{attribute 'linkalways'} 
{attribute 'no_explicit_call' := 'This FB is a CLASS and must be accessed using methods or properties'}
{attribute 'enable_dynamic_creation'}
FUNCTION_BLOCK RetrieveNodeContentValue IMPLEMENTS I_GraphVisitor, I_NodeVisitor, I_ContentVisitor
VAR
	graphUuid : T_MAXSTRING;
	nodeId : T_MAXSTRING;
	contentName : T_MAXSTRING;
	serializer : I_Serializer;
	_done : BOOL;
	_error : BOOL;
	_errorMessage : T_MAXSTRING;
END_VAR

PROPERTY PUBLIC Done : BOOL
GET
Done := _done;
END_GET
END_PROPERTY

PROPERTY PUBLIC Error : BOOL
GET
Error := _error;
END_GET
END_PROPERTY

PROPERTY PUBLIC ErrorMessage : T_MAXSTRING
GET
ErrorMessage := _errorMessage;
END_GET
END_PROPERTY

METHOD PUBLIC Initialize
VAR_INPUT
	GraphUuid : T_MAXSTRING;
	NodeId : T_MAXSTRING;
	ContentName : T_MAXSTRING;
	Serializer : I_Serializer;
END_VAR
THIS^.graphUuid := GraphUuid;
THIS^.nodeId := NodeId;
THIS^.contentName := ContentName;
THIS^.serializer := Serializer;
END_METHOD

METHOD PRIVATE LogInvalidContentNameError
VAR_INPUT
END_VAR
_errorMessage := 'Invalid Content Name';
_error := TRUE;
END_METHOD

METHOD PRIVATE LogInvalidNodeIdError
VAR_INPUT
END_VAR
_errorMessage := 'Invalid Node Id';
_error := TRUE;
END_METHOD

METHOD PRIVATE Reset
VAR_INPUT
END_VAR
_done := FALSE;
_errorMessage := '';
_error := FALSE;
END_METHOD

METHOD VisitContent
VAR_INPUT
	VisitingContent : I_Content;
END_VAR
VisitingContent.SerializeWith(serializer);
END_METHOD

METHOD VisitGraph
VAR_INPUT
	VisitingGraph : I_Graph;
END_VAR
VAR
	node : I_Node;
END_VAR
Reset();

IF NOT (VisitingGraph.Uuid = graphUuid) THEN
	RETURN;
END_IF

IF NOT VisitingGraph.Nodes.TryGetNodeById(nodeId, node) THEN
	LogInvalidNodeIdError();
	RETURN;
END_IF

node.Accept(THIS^);
END_METHOD

METHOD VisitNode
VAR_INPUT
	VisitingNode : I_Node;
END_VAR
VAR
	content : I_Content;
END_VAR
IF NOT VisitingNode.Contents.TryGetContentByName(contentName, content) THEN
	LogInvalidContentNameError();
	RETURN;
END_IF

content.Accept(THIS^);
END_METHOD

END_FUNCTION_BLOCK

(* stored: Version 1.1.0.1, ProductVersion 3.1.4024.12
   POU RetrieveNodeContentValue: Id {a2720bfd-27df-4afa-9981-101fa962f32b}, SpecialFunc None
   Folder Private: Id {07f7e8fb-406b-429c-800a-db87c2710562}
   Property Done: Id {086482da-6f85-4bc9-972c-eac3bb403e99}
   Get Get: Id {56742960-b6c7-49fb-9320-eec7c5504b00}
   Property Error: Id {9202541f-22bf-44e6-908a-fe4792893256}
   Get Get: Id {c8cddf81-ec66-4ce3-b1c2-6b686e978765}
   Property ErrorMessage: Id {0225b7bf-6149-4009-bb28-43bacb1eff25}
   Get Get: Id {260cc865-b539-4d1f-a3e4-7363d732c7b2}
   Method Initialize: Id {14fda997-e6bf-42c6-a0fc-8972feea2d05}
   Method LogInvalidContentNameError: Id {9a9aad6f-ad18-4e4e-9950-2c5635bb2fe0}
   Method LogInvalidNodeIdError: Id {4d2f526f-a648-438a-8d02-98d1a6e562bb}
   Method Reset: Id {932380b7-b4a1-46d5-91d3-91ec05f92418}
   Method VisitContent: Id {9f0a2c1b-15c8-4cbb-995b-bb40d8e7728d}
   Method VisitGraph: Id {fc5981b6-3a3b-4f96-86fa-17e119119772}
   Method VisitNode: Id {025f5b15-189e-4a15-b250-da2072a01893} *)
